// TIA Portal project "Soru1" (V15)

(* hardware
DEVICE "S7-1200 station_1"  S7-1200 Station
   slot 0: "Rack_0"  S7-1200 Rack  Rack  V1.0
   slot 1: "PLC_1"  CPU 1214C DC/DC/DC  6ES7 214-1AG40-0XB0  V4.2
*)

// ===== PLC "PLC_1"  CPU 1214C DC/DC/DC =====

VAR_GLOBAL   // PLC tag table "Default tag table"
   "Dudur" AT %I0.0 : Bool;
   "PMDyiBaslat" AT %I0.1 : Bool;
   "Cikis" AT %Q0.0 : Bool;
END_VAR

// folder: System blocks/Program resources

DATA_BLOCK "Time_H"   // DB1
{ S7_Optimized_Access := 'TRUE' }
AUTHOR : Simatic
FAMILY : IEC
NAME : IEC_TMR
VERSION : 1.0
// stored: InstanceOfName IEC_TIMER
"IEC_TIMER"
BEGIN
END_DATA_BLOCK

DATA_BLOCK "Time_L"   // DB2
{ S7_Optimized_Access := 'TRUE' }
AUTHOR : Simatic
FAMILY : IEC
NAME : IEC_TMR
VERSION : 1.0
// stored: InstanceOfName IEC_TIMER
"IEC_TIMER"
BEGIN
END_DATA_BLOCK

// folder: (top level)

ORGANIZATION_BLOCK "Main"   // OB1, LAD, ProgramCycle
TITLE = "Main Program Sweep (Cycle)"
{ S7_Optimized_Access := 'TRUE' }
VERSION : 0.1
   VAR_INPUT
      Initial_Call : Bool;   // Initial call of this OB
      Remanence : Bool;   // =True, if remanent data are available
   END_VAR
BEGIN

REGION Network 1: Zaman döngüs 2 saniye aktif 8 pasif
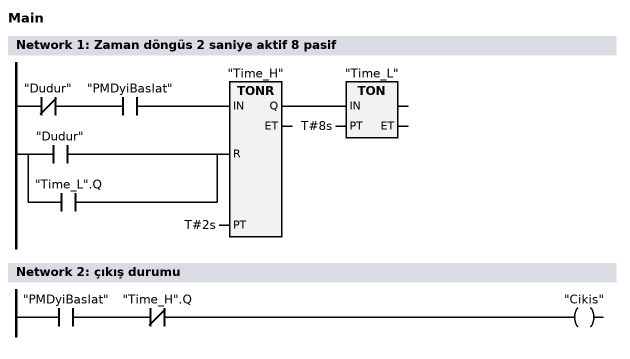
   "Time_H".TONR(IN := NOT "Dudur" AND "PMDyiBaslat", R := "Dudur" OR "Time_L".Q, PT := T#2s);
   "Time_L".TON(IN := "Time_H".Q, PT := T#8s);
END_REGION

REGION Network 2: çıkış durumu
   RUNG wire#powerrail
      Contact( "PMDyiBaslat" )
      I_Contact( "Time_H".Q )
      Coil( "Cikis" )
   END_RUNG
   // the same network as SCL:
   "Cikis" := "PMDyiBaslat" AND NOT "Time_H".Q;
END_REGION
END_ORGANIZATION_BLOCK